// TIA Portal V17 export
// export: Created 2024-10-09T16:19:46.378368Z, ExportSetting WithDefaults, DisplayName Totally Integrated Automation Portal, DisplayVersion V17, DisplayName TIA Portal Openness, DisplayVersion V17, DisplayName TIA Portal Version Control Interface, DisplayVersion V17, DisplayName STEP 7 Professional, DisplayVersion V17, DisplayName STEP 7 Safety, DisplayVersion V17, DisplayName WinCC Advanced, DisplayVersion V17
VAR_GLOBAL   // PLC tag table "Outputs"
   deckDQs AT %Q24.0 : "typeDeckControlDQ";
   mpAQs AT %Q64.0 : "typeMainPanelAQ";
   mpDQs AT %Q14.0 : "typeMainPanelDQ";
   whAQs AT %Q72.0 : "typeWheelHouseAQ";
   whDQs AT %Q80.0 : "typeWheelHouseDQ";
END_VAR
